// TIA Portal V18 export
// export: Created 2026-06-08T03:54:35.3801722Z, ExportSetting WithDefaults, DisplayName Totally Integrated Automation Portal, DisplayVersion V18, DisplayName TIA Portal Openness, DisplayVersion V18, DisplayName TIA Portal Version Control Interface, DisplayVersion V18, DisplayName STEP 7 Professional, DisplayVersion V18, DisplayName STEP 7 Safety, DisplayVersion V18, DisplayName WinCC Professional, DisplayVersion V18
ORGANIZATION_BLOCK "OB31_PID_PLC2_Bon4"   // OB31, LAD, CyclicInterrupt
{ S7_Optimized_Access := 'TRUE' }
VERSION : 0.1
// stored: AutoNumber true, IsIECCheckEnabled false, SetENOAutomatically false
   VAR_INPUT
      Initial_Call : Bool;   // Initial call of this OB
      Event_Count : Int;   // Events discarded
   END_VAR
BEGIN

REGION Network 1: PID Compact Bon 4 - call technology block
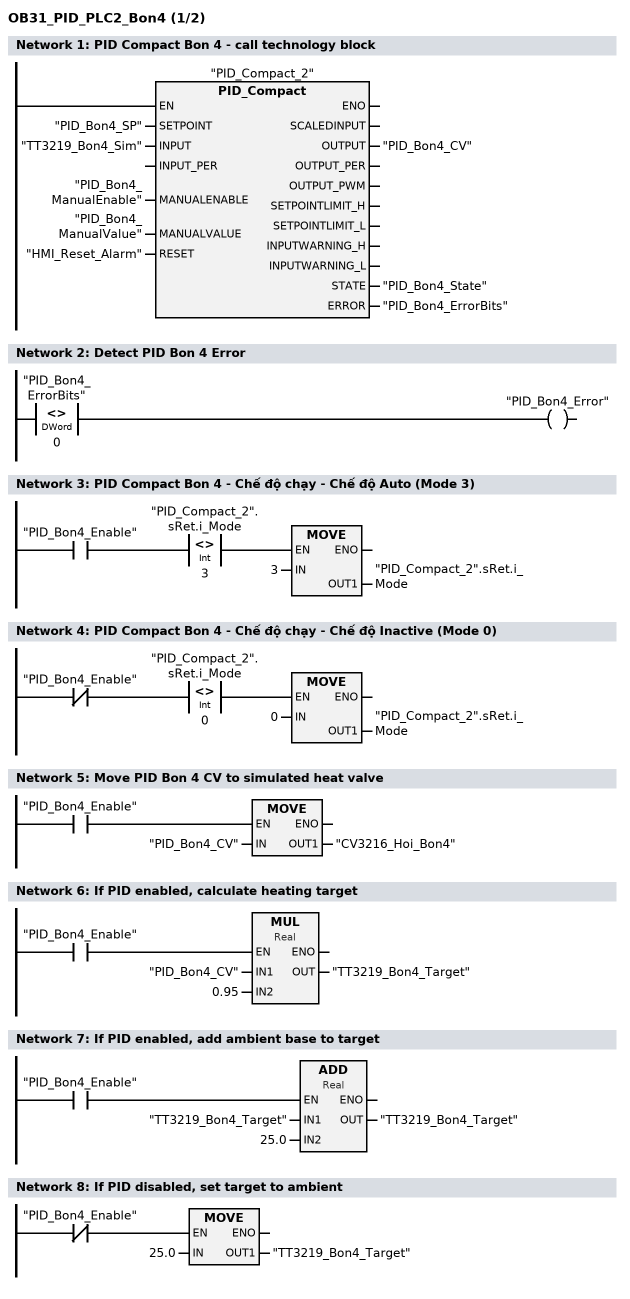
   RUNG wire#powerrail
      "PID_Compact_2".PID_Compact(Setpoint := "PID_Bon4_SP", Input := "TT3219_Bon4_Sim", Input_PER :=, ManualEnable := "PID_Bon4_ManualEnable", ManualValue := "PID_Bon4_ManualValue", Reset := "HMI_Reset_Alarm", ScaledInput =>, Output => "PID_Bon4_CV", Output_PER =>, Output_PWM =>, SetpointLimit_H =>, SetpointLimit_L =>, InputWarning_H =>, InputWarning_L =>, State => "PID_Bon4_State", Error => "PID_Bon4_ErrorBits")
   END_RUNG
   // the same network as SCL:
   "PID_Compact_2"(Setpoint := "PID_Bon4_SP",   // PID_Compact
                   Input := "TT3219_Bon4_Sim",
                   ManualEnable := "PID_Bon4_ManualEnable",
                   ManualValue := "PID_Bon4_ManualValue",
                   Reset := "HMI_Reset_Alarm",
                   Output => "PID_Bon4_CV",
                   State => "PID_Bon4_State",
                   Error => "PID_Bon4_ErrorBits");
END_REGION

REGION Network 2: Detect PID Bon 4 Error
   RUNG wire#powerrail
      { S7_Templates := "SrcType := DWord" } NE_Contact(in1 := "PID_Bon4_ErrorBits", in2 := 0)
      Coil( "PID_Bon4_Error" )
   END_RUNG
   // the same network as SCL:
   "PID_Bon4_Error" := "PID_Bon4_ErrorBits" <> 0;
END_REGION

REGION Network 3: PID Compact Bon 4 - Chế độ chạy - Chế độ Auto (Mode 3)
   RUNG wire#powerrail
      Contact( "PID_Bon4_Enable" )
      { S7_Templates := "SrcType := Int" } NE_Contact(in1 := "PID_Compact_2".sRet.i_Mode, in2 := 3)
      { S7_GenerateENO := "TRUE" } Move(in := 3, out1 => "PID_Compact_2".sRet.i_Mode)
   END_RUNG
   // the same network as SCL:
   IF "PID_Bon4_Enable" AND ("PID_Compact_2".sRet.i_Mode <> 3) THEN "PID_Compact_2".sRet.i_Mode := 3; END_IF;
END_REGION

REGION Network 4: PID Compact Bon 4 - Chế độ chạy - Chế độ Inactive (Mode 0)
   RUNG wire#powerrail
      I_Contact( "PID_Bon4_Enable" )
      { S7_Templates := "SrcType := Int" } NE_Contact(in1 := "PID_Compact_2".sRet.i_Mode, in2 := 0)
      { S7_GenerateENO := "TRUE" } Move(in := 0, out1 => "PID_Compact_2".sRet.i_Mode)
   END_RUNG
   // the same network as SCL:
   IF NOT "PID_Bon4_Enable" AND ("PID_Compact_2".sRet.i_Mode <> 0) THEN
       "PID_Compact_2".sRet.i_Mode := 0;
   END_IF;
END_REGION

REGION Network 5: Move PID Bon 4 CV to simulated heat valve
   RUNG wire#powerrail
      Contact( "PID_Bon4_Enable" )
      { S7_GenerateENO := "TRUE" } Move(in := "PID_Bon4_CV", out1 => "CV3216_Hoi_Bon4")
   END_RUNG
   // the same network as SCL:
   IF "PID_Bon4_Enable" THEN "CV3216_Hoi_Bon4" := "PID_Bon4_CV"; END_IF;
END_REGION

REGION Network 6: If PID enabled, calculate heating target
   RUNG wire#powerrail
      Contact( "PID_Bon4_Enable" )
      { S7_Templates := "SrcType := Real"; S7_GenerateENO := "TRUE" } Mul(in1 := "PID_Bon4_CV", in2 := 0.95, out => "TT3219_Bon4_Target")
   END_RUNG
   // the same network as SCL:
   IF "PID_Bon4_Enable" THEN "TT3219_Bon4_Target" := "PID_Bon4_CV" * 0.95; END_IF;
END_REGION

REGION Network 7: If PID enabled, add ambient base to target
   RUNG wire#powerrail
      Contact( "PID_Bon4_Enable" )
      { S7_Templates := "SrcType := Real"; S7_GenerateENO := "TRUE" } Add(in1 := "TT3219_Bon4_Target", in2 := 25.0, out => "TT3219_Bon4_Target")
   END_RUNG
   // the same network as SCL:
   IF "PID_Bon4_Enable" THEN "TT3219_Bon4_Target" := "TT3219_Bon4_Target" + 25.0; END_IF;
END_REGION

REGION Network 8: If PID disabled, set target to ambient
   RUNG wire#powerrail
      I_Contact( "PID_Bon4_Enable" )
      { S7_GenerateENO := "TRUE" } Move(in := 25.0, out1 => "TT3219_Bon4_Target")
   END_RUNG
   // the same network as SCL:
   IF NOT "PID_Bon4_Enable" THEN "TT3219_Bon4_Target" := 25.0; END_IF;
END_REGION

REGION Network 9: Calculate memory term: Pure * 0.99
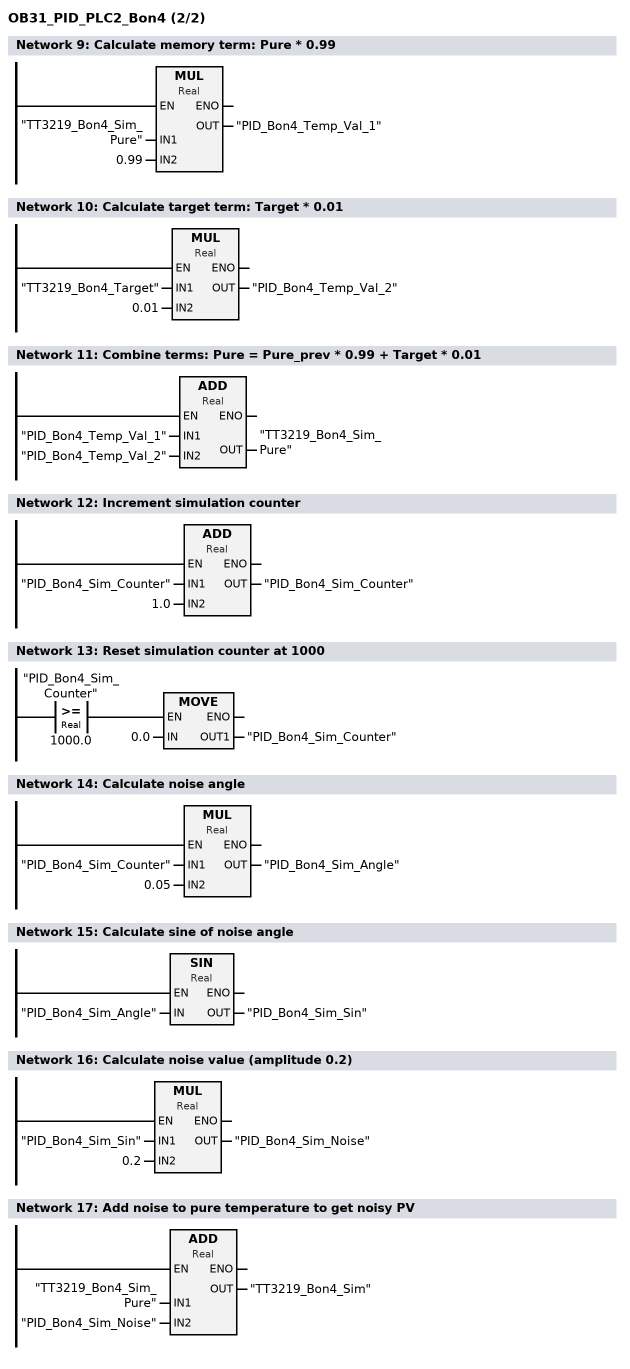
   RUNG wire#powerrail
      { S7_Templates := "SrcType := Real"; S7_GenerateENO := "TRUE" } Mul(in1 := "TT3219_Bon4_Sim_Pure", in2 := 0.99, out => "PID_Bon4_Temp_Val_1")
   END_RUNG
   // the same network as SCL:
   "PID_Bon4_Temp_Val_1" := "TT3219_Bon4_Sim_Pure" * 0.99;
END_REGION

REGION Network 10: Calculate target term: Target * 0.01
   RUNG wire#powerrail
      { S7_Templates := "SrcType := Real"; S7_GenerateENO := "TRUE" } Mul(in1 := "TT3219_Bon4_Target", in2 := 0.01, out => "PID_Bon4_Temp_Val_2")
   END_RUNG
   // the same network as SCL:
   "PID_Bon4_Temp_Val_2" := "TT3219_Bon4_Target" * 0.01;
END_REGION

REGION Network 11: Combine terms: Pure = Pure_prev * 0.99 + Target * 0.01
   RUNG wire#powerrail
      { S7_Templates := "SrcType := Real"; S7_GenerateENO := "TRUE" } Add(in1 := "PID_Bon4_Temp_Val_1", in2 := "PID_Bon4_Temp_Val_2", out => "TT3219_Bon4_Sim_Pure")
   END_RUNG
   // the same network as SCL:
   "TT3219_Bon4_Sim_Pure" := "PID_Bon4_Temp_Val_1" + "PID_Bon4_Temp_Val_2";
END_REGION

REGION Network 12: Increment simulation counter
   RUNG wire#powerrail
      { S7_Templates := "SrcType := Real"; S7_GenerateENO := "TRUE" } Add(in1 := "PID_Bon4_Sim_Counter", in2 := 1.0, out => "PID_Bon4_Sim_Counter")
   END_RUNG
   // the same network as SCL:
   "PID_Bon4_Sim_Counter" := "PID_Bon4_Sim_Counter" + 1.0;
END_REGION

REGION Network 13: Reset simulation counter at 1000
   RUNG wire#powerrail
      { S7_Templates := "SrcType := Real" } GE_Contact(in1 := "PID_Bon4_Sim_Counter", in2 := 1000.0)
      { S7_GenerateENO := "TRUE" } Move(in := 0.0, out1 => "PID_Bon4_Sim_Counter")
   END_RUNG
   // the same network as SCL:
   IF "PID_Bon4_Sim_Counter" >= 1000.0 THEN "PID_Bon4_Sim_Counter" := 0.0; END_IF;
END_REGION

REGION Network 14: Calculate noise angle
   RUNG wire#powerrail
      { S7_Templates := "SrcType := Real"; S7_GenerateENO := "TRUE" } Mul(in1 := "PID_Bon4_Sim_Counter", in2 := 0.05, out => "PID_Bon4_Sim_Angle")
   END_RUNG
   // the same network as SCL:
   "PID_Bon4_Sim_Angle" := "PID_Bon4_Sim_Counter" * 0.05;
END_REGION

REGION Network 15: Calculate sine of noise angle
   "PID_Bon4_Sim_Sin" := SIN("PID_Bon4_Sim_Angle");
END_REGION

REGION Network 16: Calculate noise value (amplitude 0.2)
   RUNG wire#powerrail
      { S7_Templates := "SrcType := Real"; S7_GenerateENO := "TRUE" } Mul(in1 := "PID_Bon4_Sim_Sin", in2 := 0.2, out => "PID_Bon4_Sim_Noise")
   END_RUNG
   // the same network as SCL:
   "PID_Bon4_Sim_Noise" := "PID_Bon4_Sim_Sin" * 0.2;
END_REGION

REGION Network 17: Add noise to pure temperature to get noisy PV
   RUNG wire#powerrail
      { S7_Templates := "SrcType := Real"; S7_GenerateENO := "TRUE" } Add(in1 := "TT3219_Bon4_Sim_Pure", in2 := "PID_Bon4_Sim_Noise", out => "TT3219_Bon4_Sim")
   END_RUNG
   // the same network as SCL:
   "TT3219_Bon4_Sim" := "TT3219_Bon4_Sim_Pure" + "PID_Bon4_Sim_Noise";
END_REGION
END_ORGANIZATION_BLOCK
